Staubli VAL3: page_viewTraj.pjx

--- page_viewTraj.pjx ---
Parameters version=s7.8.3 stackSize=5000 millimeterUnit=true
Program file=buildList.pgx
Program file=buildListFrame.pgx
Program file=editAction.pgx
Program file=goTo.pgx
Program file=insertInstr.pgx
Program file=listAdd.pgx
Program file=loadEditTraj.pgx
Program file=loadPage.pgx
Program file=main.pgx
Program file=onBackEvent.pgx
Program file=onEnterEvent.pgx
Program file=onExit.pgx
Program file=onF1Event.pgx
Program file=onF2Event.pgx
Program file=onF3Event.pgx
Program file=onF4Event.pgx
Program file=onF5Event.pgx
Program file=onF6Event.pgx
Program file=onF7Event.pgx
Program file=onF8Event.pgx
Program file=onSpaceEvent.pgx
Program file=onStart.pgx
Program file=refresh.pgx
Program file=refreshAction.pgx
Program file=refreshDynamic.pgx
Program file=refreshStatic.pgx
Program file=saveIt.pgx
Program file=selectItem.pgx
Program file=showPoint.pgx
Program file=showStatus.pgx
Program file=unSelectItem.pgx
Data file=page_viewTraj.dtx
Library alias=use path=Disk://public_temp/userPage/userPage.pjx
Library alias=pub path=Disk://public_temp/pub/pub.pjx
Library alias=data path=Disk://SaveData/SaveData.pjx

--- page_viewTraj.dtx ---
num nIndex
num nKey = 255
num nOldIndex = 2
public num nPage
num nRefresh = 13186.401
num nSelect
num nTime = 0.1
num nView
num nClockStatus
string sEvent = " 3. "
public string sItems = "test"
string sList[3]
  [0] = " 1. "
  [1] = " 2. "
  [2] = " 3. "
string sMenu[8]
  [0] = "Tool Selection"
  [2] = "Rename"
  [3] = "Paste"
  [4] = "Mark"
  [5] = "Delete"
  [6] = "Insert"
  [7] = "Save"
string sMenuUser[8]
string sMessage
string sTrajName = "test"
string sMenu8[8]
bool bButton[8]
  [0] = true
  [2] = true
  [3] = true
  [4] = true
  [5] = true
  [6] = true
  [7] = true
bool bLarge
bool bShowStatus
bool bExit
bool bTrigger
tool tTool = {fatherId=flange[0], ioLink=valve1}
frame fFather = {fatherId=world[0]}
num nBackupFrame
public string Stest[2]
string l_sltem
public string sWorkingmode[10]
  [0] = "1号石墨舟A面取片"
  [1] = "1号石墨舟A面放片"
  [2] = "1号石墨舟B面取片"
  [3] = "1号石墨舟B面放片"
  [4] = "2号石墨舟A面取片"
  [5] = "2号石墨舟A面放片"
  [6] = "2号石墨舟B面取片"
  [7] = "2号石墨舟B面放片"
  [8] = "花篮取片"
  [9] = "花篮放片"
num nSelected

--- main.pgx ---
public program main()
  local bool l_bSave
  local bool l_bOverRide
  local bool l_bContinue
  local string l_sInstruction
  local bool l_bUnreached
  local string l_sMessage
  local num l_nSize
  local num i
begin
  // INIT
  call onStart(l_bContinue)
  // LOOP UNTIL nKey=255
  do

    call refresh()
    nKey=getKey()
    call use:listevent(nKey,nIndex,sEvent)
    nView=use:nView
    nSelected=nIndex
		data:nPage_viewTraj=nIndex

    // DEFAULT FUNCTIONALITY
    switch nKey
      case 259
        // TAB
        bLarge=!bLarge
        call use:setView(bLarge)
      break
      case 263
        // backSpace rename
        call onBackEvent(l_bSave)
      break
      case 32
        // space to edit Action
        call onSpaceEvent(l_bSave)
      break
      case 271
        call onF1Event()
      break
      case 272
        //
        call onF2Event()
      break
      case 273
        //
        call onF3Event(l_bContinue,l_bSave)
      break
      case 274
        //
        call onF4Event(l_bSave)
      break
      case 275
        //
        call onF5Event()
      break
      //
      case 276
        call onF6Event(l_bSave)
      break
      case 277
        //
        call onF7Event(l_bSave)
      break
      case 278
        //
        call onF8Event(l_bSave)
      break
      case 270
        //
        call onEnterEvent(l_bSave)
      break
    endSwitch
    if workingMode()!=1 and workingMode()!=4
      call use:timerDialog("请将控制器打到手动状态或者是远程自动状态！",0)
      wait(workingMode()==1 or workingMode()==4)
    endIf
    if workingMode()==4
     // call loadPage("page/page_production")
      pub:libLoad("Disk://page/page_Production")
      call pub:main()
    endIf
    // release
    delay(0)
  until false
  cls()
  bExit=false
end

--- buildList.pgx ---
program buildList()
  local num l_nSize
  local string l_sInstruction
  local num i
  local num j
  local mdesc l_mDesc
  local num l_nTcpAction
  local string l_sEmpty
  local bool false
  local num l_nZero
  local bool l_bToStop
begin
  call use:setSizeList(17,0,21,10)
  //建立对话款
  call use:listcreate("")
// call use:selectNewField(nSelected,nIndex,nView)
  call use:listadd(sWorkingmode)
 // nIndex=data:nPage_viewTraj
  call use:selectNewField(nSelected,nIndex,nView)
  call use:listupdate(0)

    /////////////////////////////////////////////////////////////////////////////////////////////////////////////////////////////////////
    //  // INIT the list
    //  l_sEmpty=""
    //  call use:stringCopy(l_sEmpty,sList)
    //  // Build the list
    //  call trajType:getSizeItem(false,l_nSize)
    //  for i=0 to l_nSize-1
    //    if bLarge
    //      // show the instruction
    //      l_bToStop=false
    //      l_nZero=0
    //      call trajType:getTrajItem(l_tTraj,i)
    //      switch l_tTraj.nTcpAction
    //        case 1
    //          l_sInstruction="[ON],"
    //        break
    //        case 2
    //          l_sInstruction="[OFF],"
    //        break
    //        default
    //          l_sInstruction=""
    //        break
    //      endSwitch
    //      // get all the action
    //      l_sInstruction=l_sInstruction+l_tTraj.iInstr[0].sType+" "+l_tTraj.iInstr[0].sData
    //      for j=1 to size(l_tTraj.iInstr)-1
    //        l_sInstruction=l_sInstruction+","+l_tTraj.iInstr[j].sType+" "+l_tTraj.iInstr[j].sData
    //      endFor
    //      call use:typeLen(0,12,l_sInstruction,40)
    //    else
    //      call trajType:getTrajItem(l_tTraj,i)
    //      l_sInstruction=l_tTraj.comment
    //    endIf
    //    // insert the line
    //    call listAdd(toString("2",i+1)+" "+l_sInstruction)
    //  endFor
    //  // update
    //  use:bUseRefresh=true
end

--- buildListFrame.pgx ---
program buildListFrame(num x_nIndex)
  local num l_nSize
  local string l_sEvent
  local num i
  local string l_sEmpty
  local string l_sItem
begin
//  // Build the list
//  call use:setSizeList(15,0,15,11)
//  call use:listcreate("FRAME")
//  // insert all the element
//  for i=0 to size(saveData:fFrameItem)-1
//    l_sItem=toString("2",i)+" "+saveData:fFrameItem[i].sName
//    call use:listadd(l_sItem)
//  endFor
//  // update it
//  call use:listupdate(0)
//  call use:selectNewField(x_nIndex,x_nIndex,x_nIndex)
//  // leave ...
end

--- editAction.pgx ---
program editAction(bool& x_bSave[])
  local string l_sMessage
  local bool l_bOk
  local num i
  local num l_nKey
  local num l_nIndex
  local string l_sButton[2]
  local num l_nSize
  local num l_nLocal
  local string l_sEvent
  local string l_sEmpty
begin
//  // loop
//  do
//    // get the instruction
//    call trajType:getTrajItem(l_tTraj,nIndex)
//    // refresh
//    call refreshAction(l_tTraj,l_nIndex)
//    call use:typeMenu(8,"OK")
//    // get the key
//    l_nKey=get()
//    call use:listevent(l_nKey,l_nIndex,l_sEvent)
//    call use:findPos(l_sEvent,">",i)
//    i=i+3
//    switch l_nKey
//      // ENTER
//      case 270
//        // reverse video
//        call use:listcursor(l_nIndex,false)
//        switch l_nIndex
//          case 0
//            //
//            //  put a stop, after the robot reach to the point
//            //
//            l_nLocal=l_tTraj.nStop
//            call use:changeValue(l_nLocal,-1,100,i+use:nTopX,use:nView+use:nTopY+1,l_sEmpty)
//            //
//            if l_nLocal<0
//              // no stop
//              l_tTraj.toStop=false
//              l_tTraj.nStop=0
//            else
//              // stop using time
//              l_tTraj.toStop=true
//              l_tTraj.nStop=l_nLocal
//            endIf
//          break
//          case 1
//            //
//            // set TCP ON/OFF
//            //
//            // NB: 0>NONE 1>ON 2>OFF
//            call use:stringToArray("ON,OFF",sMessage)
//            if l_tTraj.nTcpAction!=0 and abs(l_tTraj.nTcpAction)<3
//              // NOTE
//              // use only absolute
//              l_tTraj.nTcpAction=abs(l_tTraj.nTcpAction)-1
//            else
//              l_tTraj.nTcpAction=0
//            endIf
//            call use:changeValue(l_tTraj.nTcpAction,0,0,i+use:nTopX,use:nView+use:nTopY+1,sMessage)
//            // give back increase by one
//            l_tTraj.nTcpAction=l_tTraj.nTcpAction+1
//          break
//          case 2,3,4
//            //
//            //  edit the instruction
//            //
//            // insert a new one
//            if l_tTraj.iInstr[l_nIndex-2].sType==""
//              call insertInstr(l_iInstr)
//              if l_sMessage!=""
//                l_tTraj.iInstr[l_nIndex-2]=l_iInstr
//              endIf
//            else
//              // delete
//              call language:message(l_sMessage,171)
//              call language:getYesNo(l_sButton)
//              // ask the yes_no question
//              call use:yes_no(l_sMessage,l_sButton,l_bOk)
//              if l_bOk
//                l_tTraj.iInstr[l_nIndex-2].sType=""
//                l_tTraj.iInstr[l_nIndex-2].sData=""
//              endIf
//            endIf
//          break
//        endSwitch
//        // save the last things
//        x_bSave=true
//        // copy back
//        call trajType:setTrajItem(l_tTraj,nIndex)
//      break
//      // SPACE
//      case 32
//        switch l_nIndex
//          call use:listcursor(l_nIndex,false)
//          case 0
//            // STOP
//            l_tTraj.toStop=!l_tTraj.toStop
//          break
//          case 1
//            // TCP
//            if l_tTraj.nTcpAction!=0
//              l_tTraj.nTcpAction=-l_tTraj.nTcpAction
//            else
//              // ON by default
//              l_tTraj.nTcpAction=1
//            endIf
//          break
//          default
//          break
//        endSwitch
//        x_bSave=true
//        // copy back
//        call trajType:setTrajItem(l_tTraj,nIndex)
//      break
//      // LEFT
//      case 264
//        // BACK
//        if nIndex>0
//          nIndex=nIndex-1
//        endIf
//      break
//      // RIGHT
//      case 268
//        // FORWARD
//        call trajType:getSizeItem(false,l_nSize)
//        if nIndex<l_nSize-1
//          nIndex=nIndex+1
//        endIf
//      break
//    endSwitch
//    // use left to go bak or escape to no validate
//  until l_nKey==278
//  // release
//  call use:nullKey(nKey)
end

--- goTo.pgx ---
program goTo(num x_nIndex, bool& x_bUnreached[])
  local bool l_bUnreached
  local num l_nIndexTool
  local tool l_tTool
  local num l_nMoveType
  local mdesc l_mDesc
begin
//  // look for not cycle mode
//  if !cycleStatus:bCycle
//    if cycleStatus:nWorkingMode==1 and isPowered()
//      // check for the index
//      if nOldIndex!=x_nIndex or (cycleStatus:nWorkingStatus!=0 and cycleStatus:nWorkingStatus!=6)
//        if !isEmpty()
//          resetMotion()
//        endIf
//        if nOldIndex!=x_nIndex
//          nOldIndex=x_nIndex
//        endIf
//      else
//        if isEmpty() and cycleStatus:nWorkingStatus==0
//          // get the data to move
//          call trajType:getTool(l_nIndexTool)
//          call tcp:getTool(l_tTool,l_nIndexTool)
//          call trajType:getTrajItem(l_tTraj,x_nIndex)
//          //
//          // use a sTemp mdesc to set the blend off
//          //
//          l_tTraj.nom_speed.blend=off
//          call trajType:goTo(l_tTool,l_tTraj.nom_speed,l_tTraj.moveType,x_bUnreached,x_nIndex)
//          call showPoint()
//        endIf
//      endIf
//    else
//      if cycleStatus:nWorkingMode!=1
//        resetMotion()
//      endIf
//    endIf
//  endIf
end

--- insertInstr.pgx ---
program insertInstr()
  local num i
  local string l_sMessage
  local num l_nIndex
  local string l_sItem
  local string l_sPath
begin
//  // create the list
//  call use:setSizeList(19,0,19,11)
//  call use:setView(false)
//  call language:message(l_sMessage,35)
//  call use:listcreate(l_sMessage)
//  // insert the action on Point
//  call use:listadd(saveData:sInstrOnPoint)
//  call use:listupdate(0)
//  // SELECT THE ITEM
//  x_iInstr.sData=""
//  do
//    i=get()
//    l_nIndex=0
//    call use:listevent(i,l_nIndex,l_sItem)
//  until i==255 or i==270
//  // update
//  x_iInstr.sType=l_sItem
//  // update
//  call saveData:getPathInstr(l_sItem,l_sPath)
//  if l_sItem!="" and i==270
//    events:libLoad(l_sPath)
//    delay(0)
//    call events:onInsert(l_sItem)
//    x_iInstr.sData=l_sItem
//  endIf
end

--- listAdd.pgx ---
program listAdd(string x_sEvent)
begin
//  // add in the queue
//  if sList!=""
//    insert(sList[size(sList)])
//  endIf
//  sList[size(sList)-1]=x_sEvent
end

--- loadEditTraj.pgx ---
program loadEditTraj(string x_sName)
  local num i
  local num l_nIndex
  local string l_sPath
begin
//  // load the traj type
//  call saveData:getPathInstr(saveData:sTrajTypeUsing,l_sPath)
//  i=trajType:libLoad(l_sPath)
//  delay(0)
//  if i!=0
//    popUpMsg("error load traj type on START "+saveData:sTrajTypeUsing+toString("",i))
//  endIf
//  // save the name
//  sTrajName=x_sName
end

--- loadPage.pgx ---
program loadPage(string x_sPage, string& x_sItems[])
// load the next page
  local num i
  local string l_sMessage
begin
//  // look if the page libload is correct
//  i=page:libLoad(x_sPage)
//  if i!=0 and i!=11
//    logMsg("INTERFACE:PAGE LIBLOAD "+x_sPage+" result "+toString("",i))
//    popUpMsg("Loading page "+x_sPage+" error CODE "+toString("",i))
//  else
//   // page:sItems=sEvent
//    call page:main()


//  endIf
end

--- onBackEvent.pgx ---
program onBackEvent(bool& x_bSave[])
  local string l_sItem
  local num i
begin
//  //
//  // rename
//  //
//  call trajType:getTrajItem(l_tTraj,nIndex)
//  if l_tTraj.comment!=""
//    i=find(sEvent,l_tTraj.comment)
//  else
//    i=len(toString("",nIndex))+3
//  endIf
//  if i!=-1
//    // clean the line
//    call use:listcursor(use:nView,false)
//    // read the name
//    call use:read(40-use:nBottomX+i-1,nView+1,l_tTraj.comment,10,false)
//    call trajType:setTrajItem(l_tTraj,nIndex)
//    call buildList()
//    x_bSave=true
//  endIf
end

--- onEnterEvent.pgx ---
program onEnterEvent(bool& x_bSave[])
  local bool l_bOk
begin
  pub:libLoad("Disk://page/page_trajectory")
  call pub:main()
end

--- onExit.pgx ---
program onExit(bool& x_bSave[])
  local string l_sMessage
  local bool l_bYes
  local frame l_fNewWorld
  local bool l_bCancel
  local string l_sButton[2]
  local num l_nResult
begin
//  // saveIt
//  if x_bSave
//    call language:message(l_sMessage,-1)
//    // get the yes_no button
//    call language:getYesNo(l_sButton)
//    // ask the question
//    call use:yes_no_cancel(l_sMessage,l_sButton,l_bYes,l_bCancel)
//    if l_bYes
//      call saveIt(x_bSave)
//    else
//      sItems[0]=""
//    endIf
//    // look for the cancel button to cancel
//    bExit=!l_bCancel
//  else
//    // exit from the page
//    bExit=true
//  endIf
//  // resetMotion
//  if !cycleStatus:bCycle
//    resetMotion()
//  endIf
//  // give back
//  // set the number
//  if size(sItems)>1
//    sItems[1]=toString("",nSelect)
//  endIf
//  // reset the show status
//  bShowStatus=false
//  //
//  call tcp:getTool(tTool,saveData:nIndexTool)
//  // give back the jog context
//  saveData:nFrameActive=nBackupFrame
//  fFather=saveData:fFrameItem[saveData:nFrameActive].fFrame
//  $jogContext(tTool,fFather,0)
end

--- onF1Event.pgx ---
program onF1Event()
  local num i
begin
//  // look if the bButton is enable
  if bButton[0]
  popUpMsg("你按下了F1按键")
  endIf
end

--- onF2Event.pgx ---
program onF2Event()
begin
//  // look if the bButton is enable
  if bButton[1]
    //
      popUpMsg("你按下了F2按键")
  endIf
end

--- onF3Event.pgx ---
program onF3Event(bool x_bContinue, bool& x_bSave[])
  local string l_sItem
  local num i
  local string l_sPage
  local string l_sEvent
  local num l_nKey
  local num l_nIndex
  local string l_sYesNo[2]
  local bool l_bValidate
  local string l_sMessage
begin
  // look if the bButton is enable
//  if bButton[2]
//    // use a list menu
//    call use:setSizeList(9,9,8,2)
//    call use:listcreate("")
//    call use:clear(0,13)
//    call use:type(9,13,sMenu[2])
//    // TOOL
//    call language:message(l_sItem,124)
//    call use:listadd(l_sItem)
//    l_sItem="Frame"
//    call use:listadd(l_sItem)
//    call use:listupdate(0)
//    // get the key
//    do
//      l_nKey=get()
//      call use:listevent(l_nKey,l_nIndex,l_sEvent)
//    until l_nKey==270 or l_nKey==255
//    // check the Enter key pressure
//    if l_nKey==270
//      switch l_nIndex
//        case 0
//          // Select the gun
//          l_sPage="Disk://kernel/page/tool"
//          call loadPage(l_sPage,l_sItem)
//          // Reload the TRAJ
//          call trajType:load(sTrajName,i)
//          // save It
//          if i!=0
//            popUpMsg("error load "+sTrajName+toString("",i))
//            x_bContinue=false
//          else
//            // logMsg
//            call trajType:setTool(saveData:nIndexTool)
//            x_bSave=true
//            //
//          endIf
//        break
//        case 1
//          // Select the Frame
//          call trajType:getFrameId(l_nIndex)
//          call buildListFrame(l_nIndex)
//          // get the Item
//          do
//            l_nKey=get()
//            call use:listevent(l_nKey,l_nIndex,l_sEvent)
//          until l_nKey==270 or l_nKey==255
//          // validate
//          if l_nKey==270
//            // TOOL advice
//            call language:message(l_sMessage,129)
//            popUpMsg(l_sMessage)
//            call use:listadd(l_sItem)
//            // question dialog for the recompute
//            call language:message(l_sMessage,227)
//            call language:getYesNo(l_sYesNo)
//            call use:yes_no(l_sMessage,l_sYesNo,l_bValidate)
//            if l_bValidate
//              // cahnge al the points into the new frame
//              call trajType:computeFrame(l_nIndex)
//            endIf
//            saveData:nFrameActive=l_nIndex
//            call trajType:setFrameId(saveData:nFrameActive)
//            x_bSave=true
//            //
//          endIf
//        break
//      endSwitch
//    endIf
//  endIf
end

--- onF4Event.pgx ---
program onF4Event(bool& x_bSave[])
  local num l_nSize
  local num i
  local num l_nTemp
begin
//  // look if the bButton is enable
//  if bButton[3]
//    //
//    // paste
//    //
//    call trajType:getSizeItem(false,l_nSize)
//    l_nTemp=nIndex+1
//    for i=0 to (l_nSize-1)
//      call trajType:getTrajItem(l_tTraj,i)
//      if find(l_tTraj.comment,"#")!=-1
//        // insert user value
//        call trajType:insertItem(i,l_nTemp)
//        if i==-1
//          return
//        else
//          // overWrite
//          l_tTraj.comment=right(l_tTraj.comment,len(l_tTraj.comment)-1)
//          call trajType:setTrajItem(l_tTraj,l_nTemp)
//          if l_nTemp<=i
//            i=i+1
//          endIf
//          l_nTemp=l_nTemp+1
//          l_nSize=l_nSize+1
//        endIf
//      endIf
//    endFor
//    // unselect ALL
//    call unSelectItem()
//    x_bSave=true
//  endIf
end

--- onF5Event.pgx ---
program onF5Event()
  local num l_nSize
begin
//  // look if the bButton is enable
//  if bButton[4]
//    //
//    //  select it
//    //
//    call selectItem(nIndex)
//    call trajType:getSizeItem(false,l_nSize)
//    // go down
//    if nIndex<l_nSize-1
//      nSelect=nIndex+1
//    endIf
//    call buildList()
//  endIf
end

--- onF6Event.pgx ---
program onF6Event(bool& x_bSave[])
  local string l_sMessage
  local num i
  local num l_nSize
  local num l_nFound
  local string l_sEvent
  local bool l_bOk
  local string l_sButton[2]
  local num l_nItem
begin
//  // look if the bButton is enable
//  if bButton[5]
//    //
//    // DELETE
//    //
//    call language:message(l_sMessage,80)
//    call language:getYesNo(l_sButton)
//    // ask the yes_no question
//    call use:yes_no(l_sMessage,l_sButton,l_bOk)
//    if l_bOk
//      // look for select one
//      call trajType:getSizeItem(false,l_nSize)
//      l_nFound=0
//      for i=0 to (l_nSize-1)
//        if l_nSize>1
//          call trajType:getTrajItem(l_tTraj,i)
//          if find(l_tTraj.comment,"#")!=-1
//            l_nFound=-1
//            // delete both normal + user
//            call trajType:deleteItem(i)
//            i=i-1
//            l_nSize=l_nSize-1
//          endIf
//        endIf
//      endFor
//      if l_nFound==0 and l_nSize>1
//        l_nItem=nIndex
//        call trajType:deleteItem(nIndex)
//        nIndex=max(nIndex-1,0)
//      endIf
//      x_bSave=true
//    endIf
//  endIf
end

--- onF7Event.pgx ---
program onF7Event(bool& x_bSave[])
  local mdesc l_mDesc
  local num l_nMoveType
  local bool l_bStop
  local num l_nTcpAction
  local num l_nItem
  local string l_sEmpty
  local num l_nDone
  local num l_nStop
begin
//  // look if the bButton is enable
//  if bButton[6]
//    //
//    // insert the user one
//    l_nItem=nIndex
//    call trajType:insertItem(nIndex,nIndex+1)
//    // empty one
//    l_sEmpty=""
//    l_bStop=false
//    l_nDone=0
//    call trajType:getTrajItem(l_tTraj,nIndex)
//    call trajType:setTrajItem(l_tTraj,nIndex+1)
//    x_bSave=true
//    nSelect=nSelect+1
//  endIf
end

--- onF8Event.pgx ---
program onF8Event(bool& x_bSave[])
  local num i
begin
//  // look if the bButton is enable
//  if bButton[7]
//    //
//    call saveIt(x_bSave)
//  endIf
end

--- onSpaceEvent.pgx ---
program onSpaceEvent(bool& x_bSave[])
begin
//  // edit the action related to the point
//  call editAction(x_bSave)
//  nSelect=nIndex
//  // refresh all
//  use:bUseRefresh=true
end

--- onStart.pgx ---
program onStart(bool& x_bResult[])
  local num i
  local num l_nIndex
  local num l_nSize
  local string l_sMessage[2]
  local bool l_bOk
begin
  cls()
  userPage()
  call use:nullKey(nKey)
  call buildList()
  call refreshStatic()
  x_bResult=true
end

--- refresh.pgx ---
program refresh()
// // page refresh
begin
  if (nKey>=270 and nKey<=278) or use:bUseRefresh==true
    cls()
    call refreshStatic()
    call buildList()
    call refreshDynamic()
    //  nIndex=data:nPage_viewTraj
    if abs(clock()-nRefresh)>nTime
      call refreshDynamic()
    endIf
  endIf
    delay(0)
end

--- refreshAction.pgx ---
program refreshAction(num x_nIndex)
  local string l_sMessage
  local string l_sTemp[3]
  local num i
begin
//  //
//  // INSTRUCTION
//  //
//  cls()
//  // create a menu to edit the action
//  call use:setSizeList(2,3,36,5)
//  call use:setView(false)
//  call use:listcreate(saveData:sTrajTypeUsing+" "+sTrajName+" "+" p. "+toString("",nIndex+1))
//  // STOP
//  call use:showBoolStatus(x_tTraj.toStop,l_sTemp)
//  call language:message(l_sMessage,174)
//  call use:strfill(l_sMessage,6,l_sMessage)
//  l_sMessage=l_sMessage+l_sTemp
//  if x_tTraj.toStop
//    // STOP
//    if round(x_tTraj.nStop)!=x_tTraj.nStop
//      l_sTemp=toString(".2",x_tTraj.nStop)+" sec"
//    else
//      l_sTemp=toString("",x_tTraj.nStop)+" sec"
//    endIf
//  else
//    // NO STOP
//    l_sTemp=""
//  endIf
//  l_sMessage=l_sMessage+"> "+l_sTemp
//  call use:listadd(l_sMessage)
//  // TCP ON OFF
//  call language:message(l_sMessage,124)
//  call use:strfill(l_sMessage,6,l_sMessage)
//  switch x_tTraj.nTcpAction
//    case 1
//      l_sTemp="[x]> ON "
//    break
//    case 2
//      l_sTemp="[x]> OFF"
//    break
//    default
//      l_sTemp="[ ]>    "
//    break
//  endSwitch
//  // ADD to the list
//  l_sMessage=l_sMessage+l_sTemp
//  call use:listadd(l_sMessage)
//  // insert all the 3 action
//  for i=0 to size(x_tTraj.iInstr)-1
//    call language:message(l_sMessage,176)
//    l_sMessage=l_sMessage+toString("",i+1)+"> "+x_tTraj.iInstr[i].sType+x_tTraj.iInstr[i].sData
//    call use:listadd(l_sMessage)
//  endFor
//  use:nView=x_nIndex
//  call use:listupdate(0)
//  // show the name
//  call language:message(l_sMessage,21)
//  l_sMessage=(l_sMessage+">"+x_tTraj.comment)
//  call use:typeLen(0,12,l_sMessage,40)
end

--- refreshDynamic.pgx ---
program refreshDynamic()
  local num i
  local string l_sInstruction
  local string l_sMessage
  local string l_sType
  local string l_sData
begin
//  // DO NOT CHANGE
  nRefresh=clock()
  use:bUseRefresh=false
//  //
//  // ADD HERE
//  //
//  // show line 12
//  call trajType:getTrajItem(l_tTraj,nIndex)
//  if bLarge
//    // show the name
//    call language:message(l_sMessage,21)
//    l_sInstruction=(l_sMessage+">"+l_tTraj.comment)
//  else
//    // select the action
//    switch l_tTraj.nTcpAction
//      case 1
//        l_sInstruction="[ON],"
//      break
//      case 2
//        l_sInstruction="[OFF],"
//      break
//      default
//      break
//    endSwitch
//    l_sType=l_tTraj.iInstr[0].sType
//    l_sData=l_tTraj.iInstr[0].sData
//    call saveInOut:replaceIO(l_sData,l_sType,l_sData)
//    l_sInstruction=l_sInstruction+l_sType+" "+l_sData
//    for i=1 to size(l_tTraj.iInstr)-1
//      if l_tTraj.iInstr[i].sType!=""
//        l_sType=l_tTraj.iInstr[i].sType
//        l_sData=l_tTraj.iInstr[i].sData
//        call saveInOut:replaceIO(l_sData,l_sType,l_sData)
//        l_sInstruction=l_sInstruction+","+l_sType+" "+l_sData
//      endIf
//    endFor
//  endIf
//  call use:typeLen(0,12,l_sInstruction,40)
//  // show the status
//  call showPoint()
end

--- refreshStatic.pgx ---
program refreshStatic()
  local string l_sMenu
  local num i
  local string l_sMessage
  local string l_sName
begin
  title("PE_Solar")
    l_sMenu="模拟,复位,,,,,,"
  // define the menu
  call use:stringToArray(l_sMenu,sMenu)
    // set the menu
  call use:setMenu(sMenu,true,2)
  call use:getMenu(sMenu,bButton)
end

--- saveIt.pgx ---
program saveIt(bool& x_bSave[])
  local string l_sMessage
  local num l_nResult
  local string l_sEmpty
begin
//  // unselect ALL
//  call unSelectItem()

//  // do the onSave trajtype
//  l_sEmpty=""
//  call trajType:onSave(l_sEmpty)
//  logMsg("[KERNEL] INTERFACE:Save the trajectory "+saveData:sTrajTypeUsing+": "+sTrajName)
//  x_bSave=false
//  sItems[0]="saved"
//  call language:message(l_sMessage,-4)
//  call use:timerDialog(l_sMessage,1)
end

--- selectItem.pgx ---
public program selectItem(num x_nIndex)
  local string l_sItem
begin
//  //
//  // select or unselect one item
//  //
//  call trajType:getTrajItem(l_tTraj,x_nIndex)
//  // check for the selected flag
//  if find(l_tTraj.comment,"#")==-1
//    l_tTraj.comment="#"+l_tTraj.comment
//  else
//    l_tTraj.comment=right(l_tTraj.comment,len(l_tTraj.comment)-1)
//  endIf
//  // set it
//  call trajType:setTrajItem(l_tTraj,x_nIndex)
end

--- showPoint.pgx ---
program showPoint()
  local point l_pPoint[2]
  local num l_nIndexTool
  local tool l_tTool
  local point l_pHere
  local num i
  local joint l_jHere
begin
//  // check for the @ position and the ! position
//  call trajType:getPoint(l_pPoint,false,nIndex)
//  call trajType:getTool(l_nIndexTool)
//  call trajType:getFrame(fFather,false)
//  call tcp:getTool(l_tTool,l_nIndexTool)
//  l_pHere=here(l_tTool,fFather)
//  // show it
//  if isEmpty() and distance(l_pHere.trsf,l_pPoint.trsf)<0.1
//    call use:type(use:nTopX,use:nTopY+1+use:nView,"@")
//  elseIf position(l_pPoint,fFather)=={0,0,0,0,0,0}
//    call use:type(use:nTopX,use:nTopY+1+use:nView,"0")
//  elseIf distance(l_pPoint.trsf,l_pHere.trsf)<10
//    call use:type(use:nTopX,use:nTopY+1+use:nView,"~")
//  elseIf !pointToJoint(l_tTool,l_jHere,l_pPoint,l_jHere)
//    call use:type(use:nTopX,use:nTopY+1+use:nView,"!")
//  else
//    call use:type(use:nTopX,use:nTopY+1+use:nView,"│")
//  endIf
end

--- showStatus.pgx ---
program showStatus()
  local joint l_jHere
  local point l_pHere
  local string l_sMessage[2]
  local tool l_tTool
begin
//  //
//  // show an dialog box with
//  // the current Joint/cartesian position
//  //
//  call tcp:getTool(l_tTool,saveData:nIndexTool)
//  if cycleStatus:nWorkingStatus>1 and cycleStatus:nWorkingStatus<5 and cycleStatus:nWorkingMode==1
//    // set a timer of x second then the message disappear ..
//    if !bTrigger
//      nClockStatus=clock()
//      bTrigger=true
//      bShowStatus=true
//    endIf
//    if clock()-nClockStatus<saveData:nTimeDialog
//      if cycleStatus:nWorkingStatus==2
//        l_jHere=herej()
//        l_sMessage="J1:"+toString("7.1",l_jHere.j1)
//        l_sMessage=l_sMessage+"  J2:"+toString("7.1",l_jHere.j2)+"#"
//        l_sMessage=l_sMessage+"J3:"+toString("7.1",l_jHere.j3)
//        l_sMessage=l_sMessage+"  J4:"+toString("7.1",l_jHere.j4)
//        //l_sMessage=l_sMessage+"  J5:"+toString("7.1",l_jHere.j5)
//        //l_sMessage=l_sMessage+"  J6:"+toString("7.1",l_jHere.j6)
//      else
//        l_pHere=here(l_tTool,fFather)
//        l_sMessage="X :"+toString("7.1",l_pHere.trsf.x)
//        l_sMessage=l_sMessage+"  Y :"+toString("7.1",l_pHere.trsf.y)
//        l_sMessage=l_sMessage+"  Z :"+toString("7.1",l_pHere.trsf.z)+"#"
//        l_sMessage=l_sMessage+"RX:"+toString("7.1",l_pHere.trsf.rx)
//        l_sMessage=l_sMessage+"  RY:"+toString("7.1",l_pHere.trsf.ry)
//        l_sMessage=l_sMessage+"  RZ:"+toString("7.1",l_pHere.trsf.rz)
//      endIf
//      call use:timerDialog(l_sMessage,0)
//    else
//      // disable it
//      bShowStatus=false
//    endIf
//  else
//    // reset it
//    if bTrigger and !cycleStatus:bCycle
//      resetMotion()
//      call showPoint()
//    endIf
//    bTrigger=false
//    bShowStatus=false
//  endIf
end

--- unSelectItem.pgx ---
program unSelectItem()
  local string l_sEvent
  local num i
  local num l_nSize
begin
//  // remove all the comments
//  call trajType:getSizeItem(false,l_nSize)
//  for i=0 to (l_nSize-1)
//    // get all the items
//    call trajType:getTrajItem(l_tTraj,i)
//    if find(l_tTraj.comment,"#")!=-1
//      // look for the select item
//      l_tTraj.comment=right(l_tTraj.comment,len(l_tTraj.comment)-1)
//      call trajType:setTrajItem(l_tTraj,i)
//    endIf
//  endFor
end
